# EPICS substitutions: epics/m-epics-eemcu/eemcuApp/Db/Sim8-extra-m1.substitutions
file "eemcu-extra.template"
{
pattern
{P,      M,    R,   PORT, ADDR, PREC, HOMEPROC}
{IOC:,   m1, m1-,   MCU1,    1, 3,    3}
}
